FUNCTION_BLOCK SOL_DIAGL (* Locally-Coupled and Clocked Diagnostics for a Solenoid *)
  (* Standard: 61499-1; Classification: Diagnostics; ApplicationDomain: Mechanisms *)
  (* Version 0.2, 2005-06-01, JHC, Holobloc Inc, Recompiled with new emitter. *)
  (* Version 0.1, 2004-10-20, JHC, Rockwell Automation, Renamed to replace old SOL_DIAGL. *)
  (* Version 0.0, 2004-09-27, JHC, Rockwell Automation, Derived from MECH2C_DIAGL. *)
  (* Compiler header: package fb.rt.mva; import fb.rt.net.*; import fb.rt.math.*; *)
  (* Compiler classdef: public class SOL_DIAGL extends FBMVCD *)
  (* Compiler Java IBM Jikes 1.06 *)
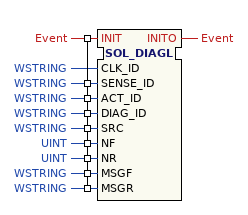
  EVENT_INPUT
    INIT WITH SENSE_ID, ACT_ID, DIAG_ID, SRC, NF, NR, MSGF, MSGR;
  END_EVENT
  EVENT_OUTPUT
    INITO;
  END_EVENT
  VAR_INPUT
    CLK_ID : WSTRING := "DIAG_CLK"; (* Diagnostic Clock Local Channel ID *)
    SENSE_ID : WSTRING; (* Sensor channel ID from Model *)
    ACT_ID : WSTRING; (* Actuator channel ID from Controller *)
    DIAG_ID : WSTRING; (* Diagnostic output channel ID *)
    SRC : WSTRING; (* Diagnostic Source ID *)
    NF : UINT; (* Forward Motion Timeout Period in CLK events *)
    NR : UINT; (* Reverse Motion Timeout Period in CLK events *)
    MSGF : WSTRING := "TIMEOUT_ADVANCING"; (* Message for fault on forward motion *)
    MSGR : WSTRING := "TIMEOUT_RETRACTING"; (* Message for fault on reverse motion *)
  END_VAR
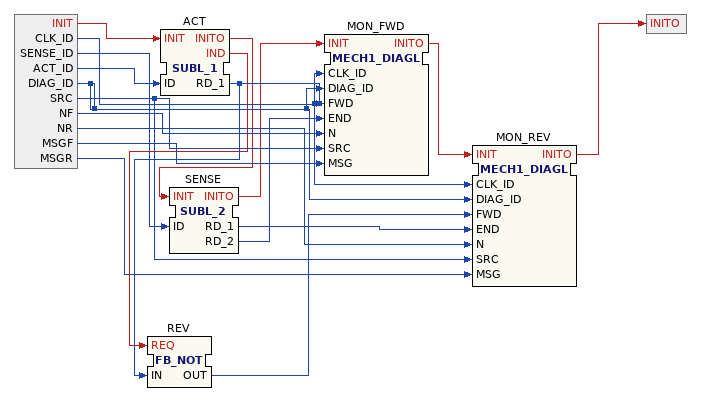
  FBS
    ACT : SUBL_1;
    SENSE : SUBL_2;
    MON_FWD : MECH1_DIAGL;
    MON_REV : MECH1_DIAGL;
    REV : FB_NOT;
  END_FBS
  EVENT_CONNECTIONS
    MON_FWD.INITO TO MON_REV.INIT;
    MON_REV.INITO TO INITO;
    INIT TO ACT.INIT;
    ACT.INITO TO SENSE.INIT;
    ACT.IND TO REV.REQ;
    SENSE.INITO TO MON_FWD.INIT;
  END_CONNECTIONS
  DATA_CONNECTIONS
    ACT_ID TO ACT.ID;
    CLK_ID TO MON_FWD.CLK_ID;
    DIAG_ID TO MON_FWD.DIAG_ID;
    ACT.RD_1 TO MON_FWD.FWD;
    NF TO MON_FWD.N;
    SRC TO MON_FWD.SRC;
    MSGF TO MON_FWD.MSG;
    CLK_ID TO MON_REV.CLK_ID;
    DIAG_ID TO MON_REV.DIAG_ID;
    NR TO MON_REV.N;
    SRC TO MON_REV.SRC;
    MSGR TO MON_REV.MSG;
    SENSE.RD_1 TO MON_REV.END;
    SENSE.RD_2 TO MON_FWD.END;
    ACT.RD_1 TO REV.IN;
    SENSE_ID TO SENSE.ID;
    REV.OUT TO MON_REV.FWD;
  END_CONNECTIONS
END_FUNCTION_BLOCK
